// SET THE CLEAN-IN-PLACE STATUS

FUNCTION SetCIP

VAR_INPUT
	
	// New CIP status
	cip : BOOL := FALSE;
	
END_VAR

VAR
	
	// Inlet enabled status
	enable : BOOL := userin.enable_in;
	
END_VAR

// I'd love a ternary operator about now...

// If in manual override
IF NOT enable THEN
	flow.in := 0;
	status.is_cip := FALSE;
	RETURN;
	
// If currently CIP -> set appropriate values	
ELSIF cip THEN
	conc.in := conc.cip;
	flow.in := flow.cip;
	
// Otherwise, set the normal values
ELSE
	conc.in := conc.normal;
	flow.in := flow.normal;
END_IF

// Update status value
status.is_cip := cip;

END_FUNCTION

(* stored: Version 1.1.0.1, ProductVersion 3.1.4024.12
   POU SetCIP: Id {70d7c6cf-0751-4d41-bb2e-68ff548ee88d}, SpecialFunc None *)
